SUBAPPLICATION Uebung_006b (* RS-Flip-Flop mit 2x IE *)
  (* Standard: 61499-2; Description: Copyright (c) 2023 Meisterschulen am Ostbahnhof This program and the accompanying materials are made available under the terms of the Eclipse Public License 2.0 which is available at https://www.eclipse.org/legal/epl-2.0/ SPDX-License-Identifier: EPL-2.0 *)
  (* Version 1.0, 2023-10-23, Franz Höpfinger, Meisterschulen am Ostbahnhof *)
  IMPORT logiBUS::io::DI::logiBUS_DI;
  IMPORT logiBUS::io::DQ::logiBUS_DO;
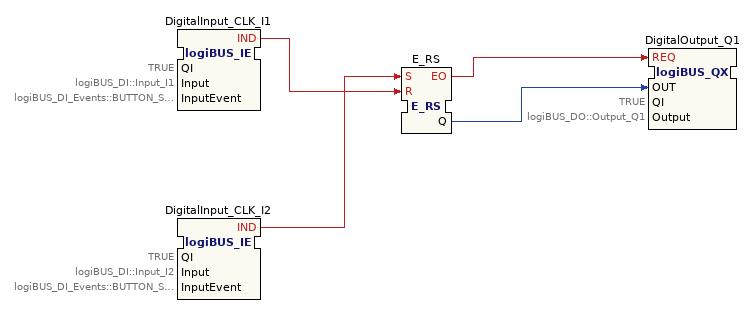
  (* Quasi wie Uebung_006 aber RS statt SR *)
  FBS
    DigitalOutput_Q1 : logiBUS::io::DQ::logiBUS_QX(QI := TRUE, Output := logiBUS_DO::Output_Q1);
    DigitalInput_CLK_I1 : logiBUS_IE(QI := TRUE, Input := logiBUS_DI::Input_I1, InputEvent := logiBUS_DI_Events::BUTTON_SINGLE_CLICK);
    DigitalInput_CLK_I2 : logiBUS_IE(QI := TRUE, Input := logiBUS_DI::Input_I2, InputEvent := logiBUS_DI_Events::BUTTON_SINGLE_CLICK);
    E_RS : iec61499::events::E_RS;
  END_FBS
  EVENT_CONNECTIONS
    DigitalInput_CLK_I2.IND TO E_RS.S;
    E_RS.EO TO DigitalOutput_Q1.REQ;
    DigitalInput_CLK_I1.IND TO E_RS.R;
  END_CONNECTIONS
  DATA_CONNECTIONS
    E_RS.Q TO DigitalOutput_Q1.OUT;
  END_CONNECTIONS
END_SUBAPPLICATION
